{attribute 'linkalways'} 
{attribute 'no_explicit_call' := 'This FB is a CLASS and must be accessed using methods or properties'}
{attribute 'enable_dynamic_creation'}
FUNCTION_BLOCK FINAL NOT_BYTE EXTENDS Node
VAR
	in : _BYTE(0);
	out : _BYTE(0);
END_VAR

METHOD PUBLIC Clone : I_Node
VAR
	pNode : POINTER TO NOT_BYTE;
END_VAR
pNode := __NEW(NOT_BYTE);
Clone := pNode^;
END_METHOD

METHOD FB_init : BOOL
VAR_INPUT
	bInitRetains : BOOL; // if TRUE, the retain variables are initialized (warm start / cold start)
	bInCopyCode : BOOL;  // if TRUE, the instance afterwards gets moved into the copy code (online change)
END_VAR
AddInput('in',THIS^.in);
AddOutput('out', THIS^.out);
END_METHOD

METHOD PROTECTED OnExecute
VAR
END_VAR
out.Value := NOT in.Value;
END_METHOD

END_FUNCTION_BLOCK

(* stored: Version 1.1.0.1, ProductVersion 3.1.4024.15
   POU NOT_BYTE: Id {c712d799-3953-4aa1-a82e-f62c9d271cf9}, SpecialFunc None
   Folder Constructor: Id {0b68fa86-1e05-4e39-a488-754e57c0b965}
   Method Clone: Id {bb0113e2-efd9-4ef9-9280-78dd656778f2}
   Method FB_init: Id {2748cfc3-bd92-4b98-89b6-66cf951d6181}
   Method OnExecute: Id {472dc778-5657-4000-8c4e-f44e89400633} *)
